PROGRAM MAIN
VAR_OUTPUT
	localTime : TIMESTRUCT;
END_VAR
VAR
	r21 : RobotA21;
	r22 : RobotA22;
	r26 : RobotA26;
END_VAR

END_PROGRAM

(* stored: Version 1.1.0.1, ProductVersion 3.1.4024.11
   POU MAIN: Id {37b3c0c4-919e-468c-8bd2-8b4a0f7831ab}, SpecialFunc None *)
